PROGRAM MAIN
VAR
	_fbPneumaticActuator : fbPneumaticActuator;
END_VAR

_fbPneumaticActuator.Manual();
_fbPneumaticActuator.SimulateInputs();

END_PROGRAM

(* stored: Version 1.1.0.1, ProductVersion 3.1.4024.2
   POU MAIN: Id {16075815-a4a8-45db-abd4-3ff94277c648}, SpecialFunc None *)
